(* IEC 61131-3 sources: RL_MAR/experiments/comparison/autoplc/results/deepseek-ai-DeepSeek-V3.2_20260508_111905/med_74, 1 file *)

(* ---- med_74_1.st ---- *)
FUNCTION_BLOCK TrafficManagementSystem
VAR_INPUT
    VehicleCount1 : INT; (* Input for vehicle count at intersection 1 *)
    VehicleCount2 : INT; (* Input for vehicle count at intersection 2 *)
    VehicleCount3 : INT; (* Input for vehicle count at intersection 3 *)
    VehicleCount4 : INT; (* Input for vehicle count at intersection 4 *)
END_VAR
VAR_OUTPUT
    TrafficLight1 : BOOL; (* Output for traffic light at intersection 1 *)
    TrafficLight2 : BOOL; (* Output for traffic light at intersection 2 *)
    TrafficLight3 : BOOL; (* Output for traffic light at intersection 3 *)
    TrafficLight4 : BOOL; (* Output for traffic light at intersection 4 *)
END_VAR

VAR
    // No internal variables needed for this simple comparison logic
END_VAR

// Process first pair: Intersection 1 and Intersection 2
IF VehicleCount1 > VehicleCount2 THEN
    TrafficLight1 := TRUE;
    TrafficLight2 := FALSE;
ELSIF VehicleCount2 > VehicleCount1 THEN
    TrafficLight1 := FALSE;
    TrafficLight2 := TRUE;
ELSE
    // Equal counts: default priority to first intersection (Intersection 1)
    TrafficLight1 := TRUE;
    TrafficLight2 := FALSE;
END_IF;

// Process second pair: Intersection 3 and Intersection 4
IF VehicleCount3 > VehicleCount4 THEN
    TrafficLight3 := TRUE;
    TrafficLight4 := FALSE;
ELSIF VehicleCount4 > VehicleCount3 THEN
    TrafficLight3 := FALSE;
    TrafficLight4 := TRUE;
ELSE
    // Equal counts: default priority to first intersection (Intersection 3)
    TrafficLight3 := TRUE;
    TrafficLight4 := FALSE;
END_IF;

END_FUNCTION_BLOCK
